// Mitsubishi GX Works2 project: dataEx02   PLC: Q02/Q02H

PROGRAM MAIN
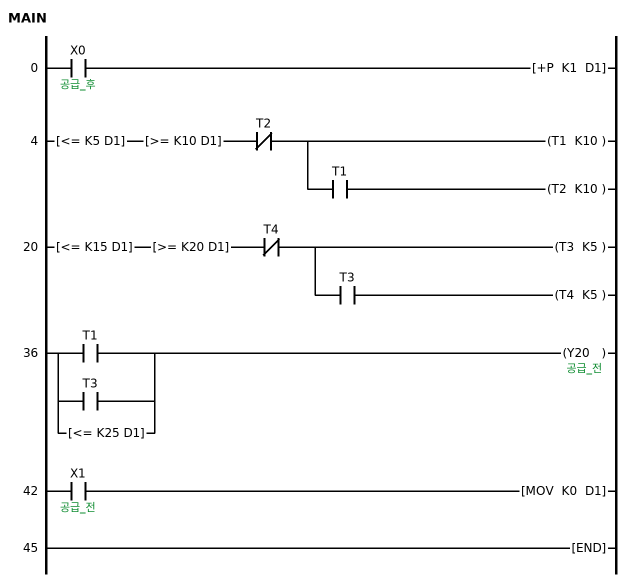
0     LD      X0  ; 공급_후
      +P      K1 D1
4     LD<=    K5 D1
      AND>=   K10 D1
      ANI     T2
      OUT     T1 K10
      AND     T1
      OUT     T2 K10
20    LD<=    K15 D1
      AND>=   K20 D1
      ANI     T4
      OUT     T3 K5
      AND     T3
      OUT     T4 K5
36    LD      T1
      OR      T3
      OR<=    K25 D1
      OUT     Y20  ; 공급_전
42    LD      X1  ; 공급_전
      MOV     K0 D1
45    END
END_PROGRAM

// device comments not shown above
X2  ; 드릴_상
X3  ; 드릴_하
X4  ; 송출_후
X5  ; 송출_전
X6  ; 배출_후
X7  ; 배출_전
X8  ; 매거진
X9  ; 비금속
X0A  ; 금속
X10  ; PB1
X11  ; PB2
X12  ; PB3
Y21  ; 공급_후
Y22  ; 드릴_하강
Y23  ; 송출_전
Y24  ; 송출_후
Y25  ; 배출_전
Y26  ; 배출_후
Y27  ; 컨베어
Y28  ; 가공드
Y29  ; 적색
Y2A  ; 황색
Y2B  ; 녹색
